TYPE TEngineCmd :
STRUCT
		SetRT : DINT;
		AutCtrl : BOOL;
		ManCtrl : BOOL;
		TurnOnMan : BOOL;
		TurnOffMan : BOOL;
		Req2RunAutCtrl : BOOL;
		ResetSUF : BOOL;
END_STRUCT
END_TYPE

(* stored: Version 1.1.0.1, ProductVersion 3.1.4024.12
   DUT TEngineCmd: Id {a181e3ef-59d9-4703-bb6c-73c44b5460e7} *)
